{attribute 'GeneratedUsingTerminal: EJ5101-0000-0016'}
{attribute addProperty BoxType "EJ5101-0000-0016"}
{attribute addProperty Id "Latch_C_validBOOL1Latch_extern_validBOOL1Set_counter_doneBOOL1Counter_underflowBOOL1Counter_overflowBOOL1Status_of_input_statusBOOL1Open_circuitBOOL1Extrapolation_stallBOOL1Status_of_input_ABOOL1Status_of_input_BBOOL1Status_of_input_CBOOL1Status_of_input_gateBOOL1Status_of_extern_latchBOOL1Sync_errorBOOL1TxPDO_StateBOOL1TxPDO_ToggleBOOL1"}
{attribute addProperty CRC "3638002371"}
{attribute addProperty Size "16"}
TYPE Status_D8D782C3 :
STRUCT
	{attribute addProperty Name "Latch_C_valid"}
	Latch_C_valid : BOOL;
	{attribute addProperty Name "Latch_extern_valid"}
	Latch_extern_valid : BOOL;
	{attribute addProperty Name "Set_counter_done"}
	Set_counter_done : BOOL;
	{attribute addProperty Name "Counter_underflow"}
	Counter_underflow : BOOL;
	{attribute addProperty Name "Counter_overflow"}
	Counter_overflow : BOOL;
	{attribute addProperty Name "Status_of_input_status"}
	Status_of_input_status : BOOL;
	{attribute addProperty Name "Open_circuit"}
	Open_circuit : BOOL;
	{attribute addProperty Name "Extrapolation_stall"}
	Extrapolation_stall : BOOL;
	{attribute addProperty Name "Status_of_input_A"}
	Status_of_input_A : BOOL;
	{attribute addProperty Name "Status_of_input_B"}
	Status_of_input_B : BOOL;
	{attribute addProperty Name "Status_of_input_C"}
	Status_of_input_C : BOOL;
	{attribute addProperty Name "Status_of_input_gate"}
	Status_of_input_gate : BOOL;
	{attribute addProperty Name "Status_of_extern_latch"}
	Status_of_extern_latch : BOOL;
	{attribute addProperty Name "Sync_error"}
	Sync_error : BOOL;
	{attribute addProperty Name "TxPDO_State"}
	TxPDO_State : BOOL;
	{attribute addProperty Name "TxPDO_Toggle"}
	TxPDO_Toggle : BOOL;
END_STRUCT
END_TYPE

(* stored: Version 1.2.0.0, ProductVersion 3.1.4024.9
   DUT Status_D8D782C3: Id {3c5c73d0-356d-417e-b69a-a65f11bf097e} *)
